Staubli VAL3: freeAdvMove.pgx

program freeAdvMove(num x_nIndex)
begin
  //setMutex(bAdvMoves)
  bAdvMoveBusy[x_nIndex]=false
  //bAdvMoves=false
end
